PROGRAM MAIN
VAR
	// trigger command execution for AWS IoT Core samples
	bGetAwsIotShadow, bPostAwsIot 	: BOOL;

	fbHttpClientAwsIot				: FB_IotHttpClient :=(sHostName := 'xyz-ats.iot.eu-central-1.amazonaws.com',
								  	bKeepAlive := FALSE, tConnectionTimeout := T#10S);
								
	fbHttpGetAwsIotShadow			: FB_TestHTTP_Get_awsIotShadow;	
	fbHttpPostAwsIot				: FB_TestHTTP_Post_awsIot;
END_VAR

// init client parameters at startup
IF NOT fbHttpClientAwsIot.bConfigured THEN 
	fbHttpClientAwsIot.stTLS.sCA := 'C:\TwinCAT\3.1\Config\Certificates\AWS\AmazonRootCA1.pem';
	fbHttpClientAwsIot.stTLS.sCert := 'C:\TwinCAT\3.1\Config\Certificates\AWS\12345678-certificate.pem.crt';
	fbHttpClientAwsIot.stTLS.sKeyFile := 'C:\TwinCAT\3.1\Config\Certificates\AWS\12345678-private.pem.key';
	fbHttpClientAwsIot.nHostPort := 8443;
END_IF

IF fbHttpClientAwsIot.bConfigured THEN
	fbHttpGetAwsIotShadow(bSend := bGetAwsIotShadow, fbClient := fbHttpClientAwsIot);
	fbHttpPostAwsIot(bSend := bPostAwsIot, fbClient := fbHttpClientAwsIot);
END_IF

fbHttpClientAwsIot.Execute();

END_PROGRAM

(* stored: Version 1.1.0.1
   POU MAIN: Id {f18145a7-ab41-4ef4-a6fc-484759a6e301}, SpecialFunc None *)
